PROGRAM EtherCAT_Diagnostic
VAR
END_VAR

END_PROGRAM

(* stored: Version 1.1.0.1, ProductVersion 3.1.4024.0
   POU EtherCAT_Diagnostic: Id {9faeb852-6688-4ea6-96af-9710c601346f}, SpecialFunc None *)
